TYPE E_SlaveArmState :
(
	SlaveArmState_Error := 1,
	SlaveArmState_Init :=2,
	SlaveArmState_SelfCheck :=3,
	SlaveArmState_Standby :=4,
	SlaveArmState_MountPanel:=5,
	SlaveArmState_PanelReady :=6,
	SlaveArmState_MountInstru :=7,
	SlaveArmState_InstruReady :=8,
	SlaveArmState_MasterSlave :=9,
	SlaveArmState_MountScope :=10,
	SlaveArmState_ScopeReady :=11,
	SlaveArmState_EndoScope :=12,
	SlaveArmState_Adjust :=13,	
	SlaveArmState_Package :=14,  		 //包装
	SlaveArmState_Cart := 15,    			 //搬运
	SlaveArmState_GravityCali := 16, 	 //重力标定
	
	SlaveArmState_totalNum :=SlaveArmState_GravityCali
);
END_TYPE

(* stored: Version 1.1.0.1, ProductVersion 3.1.4024.11
   DUT E_SlaveArmState: Id {1989848d-a357-4300-a3bc-ded8b39d8e17} *)
